// TwinCAT 3 PLC project ZK_Doc2
// Title: Doc-Test2
// Company: Lisec
// ProjectVersion: 0.4.0
// ProgramVersion: 3.1.4026.25
// libraries:
//   Doc-Test, * (Lisec)
//   Tc2_Standard, * (Beckhoff Automation GmbH)
//   Tc2_System, * (Beckhoff Automation GmbH)
// project tree:
//   POUs/ FB_Test2.TcPOU
// (motion and I/O tree: see PLC project zk_doc1)
// real-time tasks:
//   TASK PlcTask: cycle T#10ms, priority 20, ADS port 350
//   TASK PlcTask1: cycle T#10ms, priority 21, ADS port 351

// ---- POUs/FB_Test2.TcPOU
FUNCTION_BLOCK ABSTRACT FB_Test2 EXTENDS FB_Test1_Base IMPLEMENTS I_Base
VAR_INPUT
  i : INT;
END_VAR
VAR_OUTPUT
END_VAR
VAR
END_VAR

{warning 'Methodenimplementierung hinzufügen'}
/// This is a TestMethod
METHOD M_Test1 : INT
END_METHOD

METHOD M_Test2 : BOOL
VAR_INPUT
END_VAR
END_METHOD

{warning 'Eigenschaftenimplementierung hinzufügen'}
(* A Test Property with get and set*)
PROPERTY P_TestFor : BOOL
GET
END_GET
SET
END_SET
END_PROPERTY

END_FUNCTION_BLOCK
